// TIA Portal V20 export
FUNCTION_BLOCK "Clock"   // FB50, FBD
{ S7_Optimized_Access := 'FALSE' }
// stored: AutoNumber false, SetENOAutomatically false
   VAR
      Var { ExternalAccessible := 'False'; ExternalVisible := 'False'; ExternalWritable := 'False'} : "TypeVar";
      opHoRun { ExternalAccessible := 'False'; ExternalVisible := 'False'; ExternalWritable := 'False'} : Bool;
   END_VAR
   VAR_TEMP   // added for the SCL form of the ladder/FBD networks
      _w1 : Bool;
      _w2 : Bool;
   END_VAR
BEGIN

REGION Network 1: read date & time / Zeit lesen
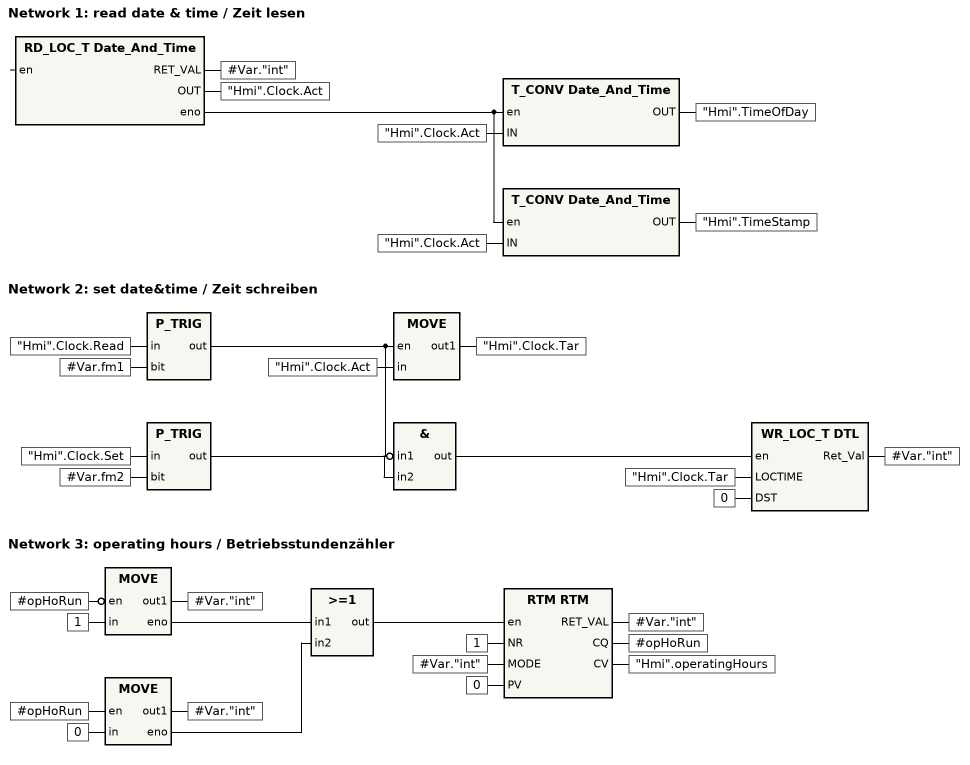
   #Var."int" := RD_LOC_T(OUT => "Hmi".Clock.Act, ENO => #_w1);
   IF #_w1 THEN
       T_CONV(IN := "Hmi".Clock.Act, OUT => "Hmi".TimeOfDay);
       T_CONV(IN := "Hmi".Clock.Act, OUT => "Hmi".TimeStamp);
   END_IF;
END_REGION

REGION Network 2: set date&time / Zeit schreiben
   #_w1 := "Hmi".Clock.Read AND NOT #Var.fm1;   // rising edge
   #Var.fm1 := "Hmi".Clock.Read;
   IF #_w1 THEN "Hmi".Clock.Tar := "Hmi".Clock.Act; END_IF;
   #_w2 := "Hmi".Clock.Set AND NOT #Var.fm2;   // rising edge
   #Var.fm2 := "Hmi".Clock.Set;
   IF NOT #_w1 AND #_w2 THEN #Var."int" := WR_LOC_T(LOCTIME := "Hmi".Clock.Tar, DST := 0); END_IF;
END_REGION

REGION Network 3: operating hours / Betriebsstundenzähler
   IF NOT #opHoRun THEN #Var."int" := 1; END_IF;
   IF #opHoRun THEN #Var."int" := 0; END_IF;
   IF NOT #opHoRun OR #opHoRun THEN
       #Var."int" := RTM(NR := 1, MODE := #Var."int", PV := 0, CQ => #opHoRun, CV => "Hmi".operatingHours);
   END_IF;
END_REGION
END_FUNCTION_BLOCK
